Fanuc KAREL source: kc00046.KL

-- PROVISIONAL review KL for V940-1; original PC SHA256 7ab24e6e2eb8de75780b19df5ec03f405bfc994fa37a0cb3bd96d0fa0c620aba
-- Incomplete behavior may be omitted. Consult companion uncertainty JSON. Do not deploy.
PROGRAM KC00046
%NOLOCKGROUP
BEGIN
  -- V9_ZERO_TABLE_METADATA_HINT layout=0002_ascii; no indexed target words; source/name/runtime held
  -- UNRESOLVED_PC offsets 5-27; opcodes 27,22,22,22,31
  -- UNRESOLVED_PC offsets 32-36; opcodes 7F
END KC00046
